PROGRAM MAIN
VAR
	b0:	INT;
	b1:	INT;
	b2: INT;
	b3: INT;
END_VAR

END_PROGRAM

(* stored: Version 1.1.0.1, ProductVersion 3.1.4024.12
   POU MAIN: Id {88b8c95c-8fd5-46d4-b8f6-98c2e094e7a7}, SpecialFunc None *)
